Staubli VAL3: start.pgx

program start()
begin
  if taskStatus("trajManage")!=-1
    taskKill("trajManage")
    wait(taskStatus("trajManage")==-1)
  endIf
  if taskStatus("motion")!=-1
    taskKill("motion")
    wait(taskStatus("motion")==-1)
  endIf
  bCycleEnd=false
  bCycle=true
  bResumeCycle=true
  taskCreate "trajManage",95,fileRead("test.txt")
  taskCreate "motion",98,trajGrind()

end
